PROGRAM POU_readSupvData
VAR
	sNetId: T_AmsNetId := SUPVams.sNetId;	// '5.30.23.91.1.1';
	nPort: T_AmsPort := SUPVams.nPort; 		// 851
	
	FB_ReadAmsValue_Fp: FB_ReadAmsValue;
	FB_ReadAmsValue_SepLevel: FB_ReadAmsValue;
	FB_ReadAmsValue_R5: FB_ReadAmsValue;
	nFpReadErrorId: UDINT;
	bFpReadError: BOOL;
	nSepLevelReadErrorId: UDINT;
	nR5ReadErrorId: UDINT;
	bSepLevelReadError: BOOL;
	bR5ReadError: BOOL;
	
	FB_ReadAmsValue_SepTempSP: FB_ReadAmsValue;
	nSepTempSPReadErrorId: UDINT;
	bSepTempSPReadError: BOOL;
	FB_ReadAmsValue_RecycleValveSP: FB_ReadAmsValue;
	bRecycleValveSPReadError: BOOL;
	nRecycleValveSPReadErrorId: UDINT;
END_VAR

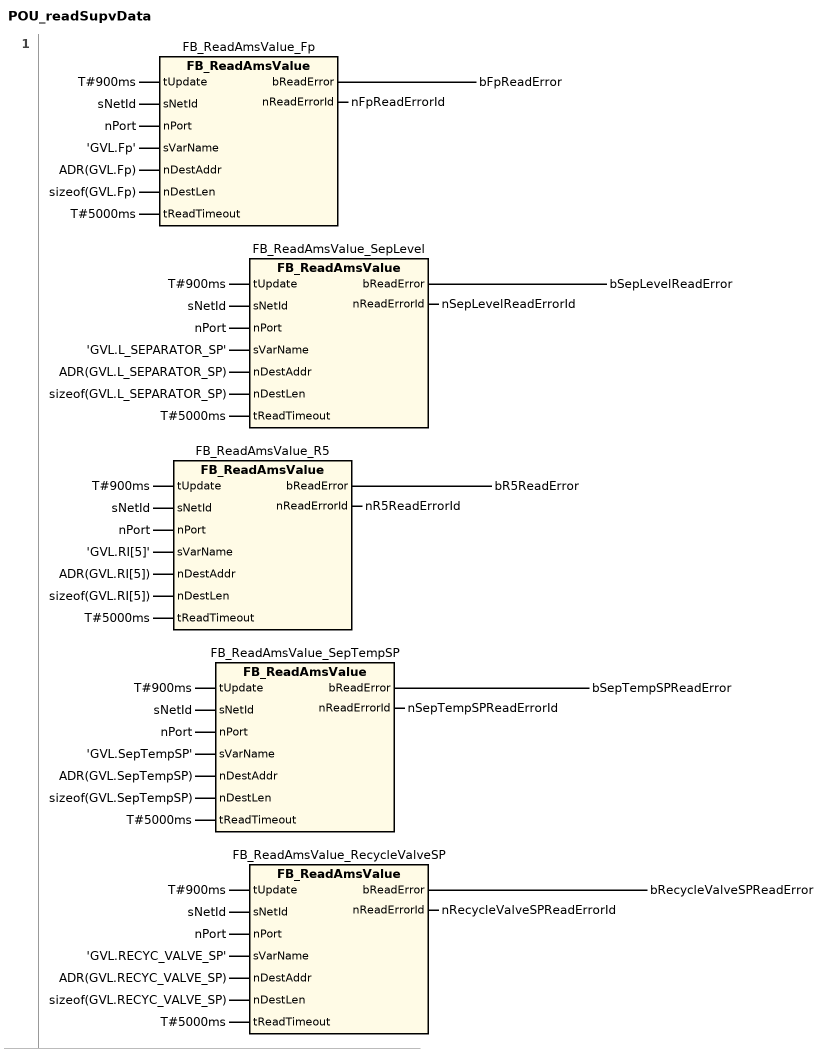
// NETWORK 1
FB_ReadAmsValue_Fp(
    tUpdate := T#900ms,
    sNetId := sNetId,
    nPort := nPort,
    sVarName := 'GVL.Fp',
    nDestAddr := ADR(GVL.Fp),
    nDestLen := sizeof(GVL.Fp),
    tReadTimeout := T#5000ms,
    nReadErrorId => nFpReadErrorId); // FB_ReadAmsValue
bFpReadError := FB_ReadAmsValue_Fp.bReadError;
FB_ReadAmsValue_SepLevel(
    tUpdate := T#900ms,
    sNetId := sNetId,
    nPort := nPort,
    sVarName := 'GVL.L_SEPARATOR_SP',
    nDestAddr := ADR(GVL.L_SEPARATOR_SP),
    nDestLen := sizeof(GVL.L_SEPARATOR_SP),
    tReadTimeout := T#5000ms,
    nReadErrorId => nSepLevelReadErrorId); // FB_ReadAmsValue
bSepLevelReadError := FB_ReadAmsValue_SepLevel.bReadError;
FB_ReadAmsValue_R5(
    tUpdate := T#900ms,
    sNetId := sNetId,
    nPort := nPort,
    sVarName := 'GVL.RI[5]',
    nDestAddr := ADR(GVL.RI[5]),
    nDestLen := sizeof(GVL.RI[5]),
    tReadTimeout := T#5000ms,
    nReadErrorId => nR5ReadErrorId); // FB_ReadAmsValue
bR5ReadError := FB_ReadAmsValue_R5.bReadError;
FB_ReadAmsValue_SepTempSP(
    tUpdate := T#900ms,
    sNetId := sNetId,
    nPort := nPort,
    sVarName := 'GVL.SepTempSP',
    nDestAddr := ADR(GVL.SepTempSP),
    nDestLen := sizeof(GVL.SepTempSP),
    tReadTimeout := T#5000ms,
    nReadErrorId => nSepTempSPReadErrorId); // FB_ReadAmsValue
bSepTempSPReadError := FB_ReadAmsValue_SepTempSP.bReadError;
FB_ReadAmsValue_RecycleValveSP(
    tUpdate := T#900ms,
    sNetId := sNetId,
    nPort := nPort,
    sVarName := 'GVL.RECYC_VALVE_SP',
    nDestAddr := ADR(GVL.RECYC_VALVE_SP),
    nDestLen := sizeof(GVL.RECYC_VALVE_SP),
    tReadTimeout := T#5000ms,
    nReadErrorId => nRecycleValveSPReadErrorId); // FB_ReadAmsValue
bRecycleValveSPReadError := FB_ReadAmsValue_RecycleValveSP.bReadError;

END_PROGRAM

(* stored: Version 1.1.0.1, ProductVersion 3.1.4024.11
   POU POU_readSupvData: Id {c8dbc9b0-45af-4c0a-8d1c-7f70f78940a5}, SpecialFunc None *)
